Fanuc KAREL source: kf00060.KL

PROGRAM KF00060
%STACKSIZE=65535
%PRIORITY=65535
%NOLOCKGROUP
VAR
I : INTEGER
J : INTEGER
X : REAL
Y : REAL
B : BOOLEAN
C : BOOLEAN
TXT : STRING[80]
TXT2 : STRING[80]
AI : ARRAY[4] OF INTEGER
BI : ARRAY[4] OF INTEGER
P : XYZWPR
JP : JOINTPOS9
PF : POSITION
STATUS : INTEGER
-- UNRESOLVED DECLARATIONS (source type spelling not recovered)
-- V1 : TYPE_0x0013 (type_u16=0x0013)
-- V2 : TYPE_0x0013 (type_u16=0x0013)
BEGIN
I=2
X=0.5
Y=1.0
-- UNRESOLVED_PC line 24 opcodes [27 22 76 23] marker_code=48
END KF00060
